DATA_BLOCK "dbArchiveControlShipping"
{ S7_Optimized_Access := 'TRUE' }
VERSION : 0.8
NON_RETAIN
"fbArchiveControlShipping"

BEGIN

END_DATA_BLOCK

